//   (this object) <-> TcCOM Objects/XTS ProcessingUnit 1/XL Part 2/XL Module 50
//     Box 62 (AT5100-0100)/DRV Commutation angle/Commutation angle <-> Data Pointer/CommutationAngle
//     Box 62 (AT5100-0100)/DRV Controlword/Controlword <-> Data Pointer/Control
//     Box 62 (AT5100-0100)/DRV Statusword/Statusword <-> Data Pointer/Status
//     Box 62 (AT5100-0100)/DRV Target torque/Target torque <-> Data Pointer/Torque
//     Box 62 (AT5100-0100)/DRV Torque actual value/Torque actual value <-> Data Pointer/ActTorque
//     Box 62 (AT5100-0100)/XFB Inputs/Data <-> Data Pointer/HallSensorValues
//   (this object) <-> TcCOM Objects/XTS ProcessingUnit 1/XL Part 2/XL Module 51
//     Box 63 (AT5100-0100)/DRV Commutation angle/Commutation angle <-> Data Pointer/CommutationAngle
//     Box 63 (AT5100-0100)/DRV Controlword/Controlword <-> Data Pointer/Control
//     Box 63 (AT5100-0100)/DRV Statusword/Statusword <-> Data Pointer/Status
//     Box 63 (AT5100-0100)/DRV Target torque/Target torque <-> Data Pointer/Torque
//     Box 63 (AT5100-0100)/DRV Torque actual value/Torque actual value <-> Data Pointer/ActTorque
//     Box 63 (AT5100-0100)/XFB Inputs/Data <-> Data Pointer/HallSensorValues
//   (this object) <-> TcCOM Objects/XTS ProcessingUnit 1/XL Part 2/XL Module 52
//     Box 64 (AT5100-0100)/DRV Commutation angle/Commutation angle <-> Data Pointer/CommutationAngle
//     Box 64 (AT5100-0100)/DRV Controlword/Controlword <-> Data Pointer/Control
//     Box 64 (AT5100-0100)/DRV Statusword/Statusword <-> Data Pointer/Status
//     Box 64 (AT5100-0100)/DRV Target torque/Target torque <-> Data Pointer/Torque
//     Box 64 (AT5100-0100)/DRV Torque actual value/Torque actual value <-> Data Pointer/ActTorque
//     Box 64 (AT5100-0100)/XFB Inputs/Data <-> Data Pointer/HallSensorValues
//   (this object) <-> TcCOM Objects/XTS ProcessingUnit 1/XL Part 2/XL Module 53
//     Box 65 (AT5100-0100)/DRV Commutation angle/Commutation angle <-> Data Pointer/CommutationAngle
//     Box 65 (AT5100-0100)/DRV Controlword/Controlword <-> Data Pointer/Control
//     Box 65 (AT5100-0100)/DRV Statusword/Statusword <-> Data Pointer/Status
//     Box 65 (AT5100-0100)/DRV Target torque/Target torque <-> Data Pointer/Torque
//     Box 65 (AT5100-0100)/DRV Torque actual value/Torque actual value <-> Data Pointer/ActTorque
//     Box 65 (AT5100-0100)/XFB Inputs/Data <-> Data Pointer/HallSensorValues
//   (this object) <-> TcCOM Objects/XTS ProcessingUnit 1/XL Part 2/XL Module 54
//     Box 66 (AT5100-0100)/DRV Commutation angle/Commutation angle <-> Data Pointer/CommutationAngle
//     Box 66 (AT5100-0100)/DRV Controlword/Controlword <-> Data Pointer/Control
//     Box 66 (AT5100-0100)/DRV Statusword/Statusword <-> Data Pointer/Status
//     Box 66 (AT5100-0100)/DRV Target torque/Target torque <-> Data Pointer/Torque
//     Box 66 (AT5100-0100)/DRV Torque actual value/Torque actual value <-> Data Pointer/ActTorque
//     Box 66 (AT5100-0100)/XFB Inputs/Data <-> Data Pointer/HallSensorValues
//   (this object) <-> TcCOM Objects/XTS ProcessingUnit 1/XL Part 2/XL Module 55
//     Box 67 (AT5100-0100)/DRV Commutation angle/Commutation angle <-> Data Pointer/CommutationAngle
//     Box 67 (AT5100-0100)/DRV Controlword/Controlword <-> Data Pointer/Control
//     Box 67 (AT5100-0100)/DRV Statusword/Statusword <-> Data Pointer/Status
//     Box 67 (AT5100-0100)/DRV Target torque/Target torque <-> Data Pointer/Torque
//     Box 67 (AT5100-0100)/DRV Torque actual value/Torque actual value <-> Data Pointer/ActTorque
//     Box 67 (AT5100-0100)/XFB Inputs/Data <-> Data Pointer/HallSensorValues
//   (this object) <-> TcCOM Objects/XTS ProcessingUnit 1/XL Part 2/XL Module 56
//     Box 68 (AT5100-0100)/DRV Commutation angle/Commutation angle <-> Data Pointer/CommutationAngle
//     Box 68 (AT5100-0100)/DRV Controlword/Controlword <-> Data Pointer/Control
//     Box 68 (AT5100-0100)/DRV Statusword/Statusword <-> Data Pointer/Status
//     Box 68 (AT5100-0100)/DRV Target torque/Target torque <-> Data Pointer/Torque
//     Box 68 (AT5100-0100)/DRV Torque actual value/Torque actual value <-> Data Pointer/ActTorque
//     Box 68 (AT5100-0100)/XFB Inputs/Data <-> Data Pointer/HallSensorValues
//   (this object) <-> TcCOM Objects/XTS ProcessingUnit 1/XL Part 2/XL Module 57
//     Box 69 (AT5100-0100)/DRV Commutation angle/Commutation angle <-> Data Pointer/CommutationAngle
//     Box 69 (AT5100-0100)/DRV Controlword/Controlword <-> Data Pointer/Control
//     Box 69 (AT5100-0100)/DRV Statusword/Statusword <-> Data Pointer/Status
//     Box 69 (AT5100-0100)/DRV Target torque/Target torque <-> Data Pointer/Torque
//     Box 69 (AT5100-0100)/DRV Torque actual value/Torque actual value <-> Data Pointer/ActTorque
//     Box 69 (AT5100-0100)/XFB Inputs/Data <-> Data Pointer/HallSensorValues
//   (this object) <-> TcCOM Objects/XTS ProcessingUnit 1/XL Part 3/XL Module 1
//     Box 74 (AT5100-0100)/DRV Commutation angle/Commutation angle <-> Data Pointer/CommutationAngle
//     Box 74 (AT5100-0100)/DRV Controlword/Controlword <-> Data Pointer/Control
//     Box 74 (AT5100-0100)/DRV Statusword/Statusword <-> Data Pointer/Status
//     Box 74 (AT5100-0100)/DRV Target torque/Target torque <-> Data Pointer/Torque
//     Box 74 (AT5100-0100)/DRV Torque actual value/Torque actual value <-> Data Pointer/ActTorque
//     Box 74 (AT5100-0100)/XFB Inputs/Data <-> Data Pointer/HallSensorValues
//   (this object) <-> TcCOM Objects/XTS ProcessingUnit 1/XL Part 3/XL Module 2
//     Box 75 (AT5100-0100)/DRV Commutation angle/Commutation angle <-> Data Pointer/CommutationAngle
//     Box 75 (AT5100-0100)/DRV Controlword/Controlword <-> Data Pointer/Control
//     Box 75 (AT5100-0100)/DRV Statusword/Statusword <-> Data Pointer/Status
//     Box 75 (AT5100-0100)/DRV Target torque/Target torque <-> Data Pointer/Torque
//     Box 75 (AT5100-0100)/DRV Torque actual value/Torque actual value <-> Data Pointer/ActTorque
//     Box 75 (AT5100-0100)/XFB Inputs/Data <-> Data Pointer/HallSensorValues
//   (this object) <-> TcCOM Objects/XTS ProcessingUnit 1/XL Part 3/XL Module 3
//     Box 76 (AT5100-0100)/DRV Commutation angle/Commutation angle <-> Data Pointer/CommutationAngle
//     Box 76 (AT5100-0100)/DRV Controlword/Controlword <-> Data Pointer/Control
//     Box 76 (AT5100-0100)/DRV Statusword/Statusword <-> Data Pointer/Status
//     Box 76 (AT5100-0100)/DRV Target torque/Target torque <-> Data Pointer/Torque
//     Box 76 (AT5100-0100)/DRV Torque actual value/Torque actual value <-> Data Pointer/ActTorque
//     Box 76 (AT5100-0100)/XFB Inputs/Data <-> Data Pointer/HallSensorValues
//   (this object) <-> TcCOM Objects/XTS ProcessingUnit 1/XL Part 3/XL Module 4
//     Box 77 (AT5100-0100)/DRV Commutation angle/Commutation angle <-> Data Pointer/CommutationAngle
//     Box 77 (AT5100-0100)/DRV Controlword/Controlword <-> Data Pointer/Control
//     Box 77 (AT5100-0100)/DRV Statusword/Statusword <-> Data Pointer/Status
//     Box 77 (AT5100-0100)/DRV Target torque/Target torque <-> Data Pointer/Torque
//     Box 77 (AT5100-0100)/DRV Torque actual value/Torque actual value <-> Data Pointer/ActTorque
//     Box 77 (AT5100-0100)/XFB Inputs/Data <-> Data Pointer/HallSensorValues
//   (this object) <-> TcCOM Objects/XTS ProcessingUnit 1/XL Part 3/XL Module 46
//     Box 72 (AT5100-0100)/DRV Commutation angle/Commutation angle <-> Data Pointer/CommutationAngle
//     Box 72 (AT5100-0100)/DRV Controlword/Controlword <-> Data Pointer/Control
//     Box 72 (AT5100-0100)/DRV Statusword/Statusword <-> Data Pointer/Status
//     Box 72 (AT5100-0100)/DRV Target torque/Target torque <-> Data Pointer/Torque
//     Box 72 (AT5100-0100)/DRV Torque actual value/Torque actual value <-> Data Pointer/ActTorque
//     Box 72 (AT5100-0100)/XFB Inputs/Data <-> Data Pointer/HallSensorValues
//   (this object) <-> TcCOM Objects/XTS ProcessingUnit 1/XL Part 3/XL Module 47
//     Box 73 (AT5100-0100)/DRV Commutation angle/Commutation angle <-> Data Pointer/CommutationAngle
//     Box 73 (AT5100-0100)/DRV Controlword/Controlword <-> Data Pointer/Control
//     Box 73 (AT5100-0100)/DRV Statusword/Statusword <-> Data Pointer/Status
//     Box 73 (AT5100-0100)/DRV Target torque/Target torque <-> Data Pointer/Torque
//     Box 73 (AT5100-0100)/DRV Torque actual value/Torque actual value <-> Data Pointer/ActTorque
//     Box 73 (AT5100-0100)/XFB Inputs/Data <-> Data Pointer/HallSensorValues
//   (this object) <-> TcCOM Objects/XTS ProcessingUnit 1/XL Part 3/XL Module 5
//     Box 78 (AT5100-0100)/DRV Commutation angle/Commutation angle <-> Data Pointer/CommutationAngle
//     Box 78 (AT5100-0100)/DRV Controlword/Controlword <-> Data Pointer/Control
//     Box 78 (AT5100-0100)/DRV Statusword/Statusword <-> Data Pointer/Status
//     Box 78 (AT5100-0100)/DRV Target torque/Target torque <-> Data Pointer/Torque
//     Box 78 (AT5100-0100)/DRV Torque actual value/Torque actual value <-> Data Pointer/ActTorque
//     Box 78 (AT5100-0100)/XFB Inputs/Data <-> Data Pointer/HallSensorValues
//   (this object) <-> TcCOM Objects/XTS ProcessingUnit 1/XL Part 3/XL Module 6
//     Box 79 (AT5100-0100)/DRV Commutation angle/Commutation angle <-> Data Pointer/CommutationAngle
//     Box 79 (AT5100-0100)/DRV Controlword/Controlword <-> Data Pointer/Control
//     Box 79 (AT5100-0100)/DRV Statusword/Statusword <-> Data Pointer/Status
//     Box 79 (AT5100-0100)/DRV Target torque/Target torque <-> Data Pointer/Torque
//     Box 79 (AT5100-0100)/DRV Torque actual value/Torque actual value <-> Data Pointer/ActTorque
//     Box 79 (AT5100-0100)/XFB Inputs/Data <-> Data Pointer/HallSensorValues
//   (this object) <-> TcCOM Objects/XTS ProcessingUnit 1/XL Part 3/XL Module 7
//     Box 80 (AT5100-0100)/DRV Commutation angle/Commutation angle <-> Data Pointer/CommutationAngle
//     Box 80 (AT5100-0100)/DRV Controlword/Controlword <-> Data Pointer/Control
//     Box 80 (AT5100-0100)/DRV Statusword/Statusword <-> Data Pointer/Status
//     Box 80 (AT5100-0100)/DRV Target torque/Target torque <-> Data Pointer/Torque
//     Box 80 (AT5100-0100)/DRV Torque actual value/Torque actual value <-> Data Pointer/ActTorque
//     Box 80 (AT5100-0100)/XFB Inputs/Data <-> Data Pointer/HallSensorValues
//   (this object) <-> TcCOM Objects/XTS ProcessingUnit 1/XL Part 3/XL Module 8
//     Box 81 (AT5100-0100)/DRV Commutation angle/Commutation angle <-> Data Pointer/CommutationAngle
//     Box 81 (AT5100-0100)/DRV Controlword/Controlword <-> Data Pointer/Control
//     Box 81 (AT5100-0100)/DRV Statusword/Statusword <-> Data Pointer/Status
//     Box 81 (AT5100-0100)/DRV Target torque/Target torque <-> Data Pointer/Torque
//     Box 81 (AT5100-0100)/DRV Torque actual value/Torque actual value <-> Data Pointer/ActTorque
//     Box 81 (AT5100-0100)/XFB Inputs/Data <-> Data Pointer/HallSensorValues

CONFIGURATION PlanarTrackMovement_1
    RESOURCE PLC ON TwinCAT3
        TASK PlcTask(INTERVAL := T#2ms, PRIORITY := 20);
        PROGRAM MAIN WITH PlcTask : MAIN;
    END_RESOURCE
END_CONFIGURATION

// ---- DUTs/E_EcState.TcDUT
{attribute 'qualified_only'}
{attribute 'strict'}
{attribute 'to_string'}
TYPE E_EcState :
(
	InitNoCom_Fault := 0,
	Init := 1,
	Preop := 2,
	Boot := 3,
	SafeOP := 4,
	Op_Ready := 8
)UINT := InitNoCom_Fault ;
END_TYPE

// ---- DUTs/E_MergeMode.TcDUT
{attribute 'qualified_only'}
{attribute 'strict'}
TYPE E_MergeMode :
(
	BlockedWait := 0,
	Follow := 1,
	Lead := 2
);
END_TYPE

// ---- DUTs/E_SwitchOpMode.TcDUT
{attribute 'qualified_only'}
//{attribute 'strict'}
TYPE E_SwitchOpMode :
(
  DivertSpecifiedCount	:= 0,
  DivertAll	:= 1
);
END_TYPE

// ---- DUTs/E_TrackNum.TcDUT
{attribute 'qualified_only'}
{attribute 'strict'}
TYPE e_TrackNum :
	(
	Main   :=1,
	Small  :=2,
	Big    :=3
	);	
END_TYPE

// ---- DUTs/MoverSort.TcDUT
TYPE MoverSort :
STRUCT
	MoverNumber 	: UDINT;
	TrackID  		: PlanarTrackOTCID;
	MoverPos 		: LREAL;
	MoverTrackNr 	: UDINT;
END_STRUCT
END_TYPE

// ---- DUTs/ST_Color_Code.TcDUT
TYPE ST_Color_Code :
STRUCT
	Pattern : UINT;
	Red :USINT;
	Green: USINT;
	Blue : USINT; 
END_STRUCT
END_TYPE

// ---- DUTs/ST_DivertConfig.TcDUT
TYPE ST_DivertConfig :
STRUCT
 	SwitchOpMode         						: E_SwitchOpMode;
	IntervalToDivert							: UDINT := 1;
	MaxAllowedDivertCount						: UDINT := 0;
	CurrentFunctionCoeffA						: LREAL := 0.5;
	CurrentFunctionCoeffB						: LREAL := 0.3;
	CurrentFunctionCoeffC						: LREAL := 5.5;
END_STRUCT
END_TYPE;

// ---- DUTs/ST_MergeConfig.TcDUT
TYPE ST_MergeConfig :
STRUCT
	gapStart: LREAL := 5600;
	gapLength: LREAL := 2000;
	moverInFront: UDINT;
	mover1FollowDist: LREAL;
	followSyncPos: LREAL;
	masterSyncPos: LREAL;
	masterPosAtSync: LREAL;
	followerPosAtSync: LREAL;
END_STRUCT
END_TYPE;

// ---- DUTs/ST_MoverConfig.TcDUT
TYPE ST_MoverConfig EXTENDS ST_MoveOnTrackOptions:
STRUCT
	Velo			: LREAL := 1500;
	Accel			: LREAL := 4000;
	Decel			: LREAL := 4000;
	Jerk			: LREAL := 16000;
	VeloComp		: LREAL := 200;
	MoverGap		: LREAL := 900;
END_STRUCT
END_TYPE

// ---- DUTs/ST_PlanarTrackConfig.TcDUT
TYPE ST_PlanarTrackConfig :
STRUCT
	TrackIndex					: E_TrackNum;
	MCTrack						: CDT_MCTOPLC_PLANAR_TRACK;
END_STRUCT
END_TYPE

// ---- DUTs/ST_StaticSectorStatus.TcDUT
TYPE ST_StaticSectorStatus :
STRUCT
	MoverIsOnSector			: BOOL;
	MoverCountOnSector		: UDINT;
	MoverEnteredSector		: Tc2_Standard.R_TRIG;
	MoverExitedSector		: Tc2_Standard.F_TRIG;
	SectorLength				: LREAL;
	MoverDistanceFromEnd	: LREAL;
END_STRUCT
END_TYPE

// ---- DUTs/ST_SwitchConfig.TcDUT
TYPE ST_SwitchConfig :
STRUCT
	MagnetStartPosition				    	    : LREAL := 9850; // mm
	MagnetEndPosition				    	    : LREAL := 10600; // mm
	OnInnerLoopOffMagnetPosn					: LREAL	:= 170; //mm
	SwitchCurrentNominal						: LREAL := 5.8; // A (See function for computation)
	CurrentMultFactor							: LREAL := 1310; // Scaling factor for 10V output=25.0A
    UseNominalCurrentVeloSetpoints              : BOOL;
    UseNominalPositionCoeff			            : BOOL := TRUE;
 	DivertConfig	       						: ST_DivertConfig;
END_STRUCT
END_TYPE;

// ---- DUTs/ST_SwitchStatus.TcDUT
TYPE ST_SwitchStatus :
STRUCT
 	MagnetValue		        AT%Q* 	: INT;
	MagnetEnabled     	        	: BOOL;
    CurrentOutputActual             : LREAL;
    CurrentTheorOutputMax           : LREAL;
	CurrentActualOutput				: LREAL;
    PosnCurrentCoeff                : LREAL;
	ShuttleCountAtDivertTrig		: UDINT;
	ShuttleQueueCount				: UDINT;
	ShuttleCountOnShortcut			: UDINT;
END_STRUCT
END_TYPE

// ---- XlMover/DUTs/DUT.TcDUT
TYPE ST_XtsCommandFeedback :
STRUCT
		(* Returns wether the execution of the method is done. *)
		IsDone : BOOL;
		(* Returns wether the execution of the method is busy. *)
		IsBusy : BOOL;
		(* Returns wether the execution of the method is busy. *)
		HasError : BOOL;
		(* Returns the HRESULT to the call. *)
		{attribute 'GUID' := '18071995-0000-0000-0000-000000000019'}
		{attribute 'GlobalType'}
		HRESULT : GLOBAL.HRESULT;
	END_STRUCT
END_TYPE

// ---- GVLs/GVL_Mc.TcGVL

VAR_GLOBAL PERSISTENT
	nNumMovers			: UINT := 16;
END_VAR


VAR_GLOBAL CONSTANT
	nMoverCount					: UINT := 16;
	nTrackCount					: UINT := 3;
	gciNumStations 				: UINT := 3;
	XtsShortcutOid				: otcid := 16#01010480 ;
	XtsOutterLoopOid 			: otcid := 16#01010490;
END_VAR

VAR_GLOBAL
	//Track_BigCircle		: 	MC_PlanarTrack; 	
	//Track_MainCircle	: 	MC_PlanarTrack;
 	//Track_SmallCircle	: 	MC_PlanarTrack;
	
	MC_Tracks    		:	ARRAY[1..nTrackCount] OF MC_PlanarTrack;
	MC_Trackfeedback	:	ARRAY[1..nTrackCount] OF MC_PlanarFeedback;
	TrackTrail 			:	MC_PlanarTrackTrail;
	
	fbXtsEnvironment			: 	FB_XtsEnvironment;
	ipXlMover 					: 	I_XtsXlMover1;
	ipXtsProcessingUnit			:   I_XtsProcessingUnit1;
	cmdFeedback					: 	XtsCommandFeedback;
	fbMover				:	ARRAY[1..nMoverCount] OF FB_Mover;
	iMover				:	ARRAY[1..nMoverCount] OF I_Mover;
	//fbPlanarMover		:	ARRAY[1..nNumMaxMovers] OF FB_PlanarMover;
	MoverFeedback		:	ARRAY[1..nMoverCount] OF MC_PlanarFeedback;
	aStopPositions : ARRAY [1..nMoverCount] OF LREAL;// := [2400, 1700, 1000, 300];
	
	
	Mover				:	ARRAY[0..nMoverCount] OF MoverSort;
	
	HWStart		AT%I* : BOOL;
	HWStop		AT%I* : BOOL;	
	StartLight 	AT%Q* : BOOL;
	StopLight	AT%Q* : BOOL;
	
	sGraphCalciFrame : T_MaxString := 'https://www.desmos.com/calculator';
END_VAR

// ---- XlMover/ITFs/I_Mover.TcIO

INTERFACE I_Mover

METHOD CycleUpdate : BOOL
VAR_INPUT
END_VAR
END_METHOD

PROPERTY distToEndOfTrack : Lreal
GET
END_GET
END_PROPERTY

METHOD Init : BOOL
VAR_INPUT
	XtsMover:  I_XtsXlMover1;
	XtsProcessingUnit :  I_XtsProcessingUnit1;
END_VAR
END_METHOD

METHOD JoinNearestTrack : BOOL


VAR

END_VAR
END_METHOD

METHOD LeaveSystemAt : BOOL
VAR_INPUT
	ConnectionOut: REFERENCE TO MC_PlanarTrackConnectionOut;	
END_VAR
END_METHOD

METHOD MoveOnTrack : BOOL
VAR_INPUT
	track: REFERENCE TO MC_PlanarTrack;	
	targetPos: LREAL;
	gap : LREAL; 
	velo : LREAL; 
END_VAR
END_METHOD

PROPERTY MoverOTCID : OTCID
GET
END_GET
SET
END_SET
END_PROPERTY

PROPERTY MoverStopped : BOOL
GET
END_GET
SET
END_SET
END_PROPERTY

PROPERTY P_Dynamics : REFERENCE TO DynamicConstraint_PathXY;
GET
END_GET
END_PROPERTY

PROPERTY P_IsInitialized : bool
GET
END_GET
END_PROPERTY

PROPERTY P_PlanarFeedback : REFERENCE TO MC_PlanarFeedback
GET
END_GET
END_PROPERTY

PROPERTY P_PlanarMover :   REFERENCE TO  MC_PlanarMover
GET
END_GET
END_PROPERTY

PROPERTY P_SyncFeedback :  REFERENCE TO MC_PlanarFeedbackGearInPosOnTrackWithMasterMover
GET
END_GET
END_PROPERTY

PROPERTY P_TargetTrack : UDINT
GET
END_GET
SET
END_SET
END_PROPERTY

PROPERTY Rework : BOOL
GET
END_GET
SET
END_SET
END_PROPERTY

METHOD SyncToOtherMover : Bool
VAR_INPUT
	masterSyncPos : LREAL; // Position on the master track
	followerSyncPos : LREAL; // position on the follower track
	PlanarMoverToFollow: REFERENCE TO Tc3_Mc3PlanarMotion.MC_PlanarMover;
	masterTrack : REFERENCE TO Tc3_Mc3PlanarMotion.MC_PlanarTrack; 
	followerTrack : REFERENCE TO Tc3_Mc3PlanarMotion.MC_PlanarTrack; 
	velo :  REFERENCE TO LREAL; 
END_VAR
END_METHOD

METHOD  UpdateXtsTrack
VAR_INPUT
END_VAR
VAR

END_VAR
END_METHOD

PROPERTY XlProcessingUnit : I_XtsProcessingUnit1
GET
END_GET
END_PROPERTY

PROPERTY XtsComFeed : REFERENCE TO  XtsCommandFeedback
GET
END_GET
END_PROPERTY

PROPERTY XtsXlMover :  I_XtsXlMover1
GET
END_GET
END_PROPERTY

END_INTERFACE

// ---- POUs/MAIN.TcPOU
PROGRAM MAIN
VAR

	bAllDone		: BOOL;
	bStopSequence	: BOOL;
	HMI_StopCmd		: BOOL;
	
	nCase 		: INT;
	nMoveState		: ARRAY[1..nMoverCount] OF INT;
	

	
	nForCounter: UDINT;
	M,N,T,Tr : UINT;
//	slowDynamics: DynamicConstraint_PathXY;
	haltDynamics : DynamicConstraint_PathXY;
	stopAndWait : ARRAY[1..GVL_Mc.nMoverCount] OF TON; 
	waitForGapParkPos: LREAL := 3500;
	// Magnet
	MagnetValue AT%Q*: INT;
	MagnetFdbkValue AT%I* : INT;
	bMagnetOn : BOOL;	

	Init : BOOL ; 	
	
	IsMoverCommandedInShortcut: BOOL;
	IsMoverInBlockingArea: BOOL;
	nActStopPos: UINT := 1;
	Fp_error : R_Trig;

	Switch : BOOL;
	WithoutSwitch : BOOL := TRUE;
	SwtichOnly: BOOL;
	
	MoverStop 	AT%I* :BOOL;
	MoverStopDone AT%Q*		: BOOL;
	Info 		AT%Q*: BOOL;
	Operating	AT%Q*: BOOL;
	Process		AT%Q*: BOOL;
	Fault		AT%Q*: BOOL;
	Emergency	AT%Q*: BOOL;
	
	Voltage1 AT%I*: UDINT;
	Voltage2 AT%I*: UDINT;
	
	
	TcRestart : TC_Restart;
	Restart : BOOL;
	busy : BOOL;
	rt_InitStart : R_TRIG;
	rt_InitStop : R_TRIG;
	bStartSequence: BOOL;
	
	FP_Counter : r_trig;
	Switchcounter : DINT;
	test : LREAL;
	Horntimer : tp; 
	R_trigHorn : R_trig;
	
	TestPowerMat : BOOL := TRUE;
	StopTime : TIME := T#1S;
	StopTimer :ARRAY[1..nMoverCount] OF ton;
	StartTimer :ARRAY[1..nMoverCount] OF BOOL;
	
	
	MoverPos :ARRAY[1..nMoverCount] OF PositionXYC;
	ArcLength :ARRAY[1..nMoverCount] OF LREAL;
	TrackPos :ARRAY[1..nMoverCount] OF ARRAY[1..nMoverCount] OF PositionXYC;
	
	//searchGap : F_SearchTheBigTrackForAHole; 
	aMoverTrack : ARRAY[1..nMoverCount] OF Global.OTCID;
	FirstMoverTrackPos : LREAL;
	MoverGap : LREAL;
	FTrigTrackCount : F_Trig;
	MoverNo  : UDINT;
	stMoverConfigSlow	: ST_MoverConfig;
	stMoverConfigNormal : ST_MoverConfig;
	stMoverConfigFast  : ST_MoverConfig;
	stMoverCfgAggressive : ST_MoverConfig;
	stMoverCfgHalt : ST_MoverConfig;
	
	stMergeConfig		 : ST_MergeConfig;
	SwitchConfig		 : ST_SwitchConfig;
	
	SwitchStatus 		  : ST_SwitchStatus;

	ModuleState1 AT%I*: E_EcState;
	ModuleState2 AT%I*: E_EcState;
	ModuleState3 AT%I*: ARRAY[0..2] OF E_EcState;
	
	MessageTrigger : ARRAY[1..20] OF R_trig;
	
	//========= Merge =========================================
	
	SwitchParkPos : LREAL := 3500;
	nextMoverForSwitch: UDINT :=1;
	moverInSwitchDoNotSendAnother: BOOL;
	trapError: BOOL;
	trapErrorID: UDINT;
	moverWithFault: UDINT;
	stepWithFault: INT;
	
	followSyncPos: LREAL;
	masterSyncPos: LREAL;
	masterPosAtSync: LREAL;
	followerPosAtSync: LREAL;
	moverInFront: UDINT;
	gapStart: LREAL := 8500; //5600
	gapLength: LREAL := 2200; //1800
	fbTrackobject : FB_TrackObject;
	getList: BOOL;
	directMerge: BOOL;
	mergeNotPossible: BOOL;
	
	endOfBigTrack : LREAL; 
	endOfSmallTrack : LREAL; 
	endOfMainTrack : LREAL; 
	followerToEndOfTrack: LREAL;
	leaderToEndofTrack: LREAL;
	distToMoverInFront: LREAL;
END_VAR


// =====================
// Initalize XTS Utility
GVL_MC.fbXtsEnvironment.Init(GVL_MC.cmdFeedback);
IF NOT GVL_MC.cmdFeedback.IsDone THEN
	RETURN;
END_IF
//*****************************************************
Emergency :=  MoverStop;

Operating := NOT  MoverStop;

//================== Check Voltage=====================================================
R_trigHorn(clk := Voltage1< 250000 );
//Horntimer(in:= ( R_trigHorn.Q ) , PT:= T#2S,Q=> info);
IF R_trigHorn.Q THEN
	ADSLOGSTR(msgCtrlMask:= ADSLOG_MSGTYPE_LOG , msgFmtStr:= 'Module Voltage Fault ' , strArg:= '');
END_IF 
//=================== Check State of Modules===========================================

MessageTrigger[1](clk:=ModuleState1 <> 8 AND nCASE> 0);
IF MessageTrigger[1].Q THEN
	ADSLOGSTR(msgCtrlMask:= ADSLOG_MSGTYPE_LOG , msgFmtStr:= 'Module Fault Line 1 %s' , strArg:= TO_STRING(ModuleState1));
END_IF

MessageTrigger[2](clk:=ModuleState2 <> 8 AND nCASE> 0);
IF MessageTrigger[2].Q THEN
	ADSLOGSTR(msgCtrlMask:= ADSLOG_MSGTYPE_LOG , msgFmtStr:= 'Module Fault Line 2 %s ' , strArg:= TO_STRING(ModuleState2));
END_IF

MessageTrigger[3](clk:=ModuleState3[0] <> 8 AND nCASE> 0);
IF MessageTrigger[3].Q THEN
	ADSLOGSTR(msgCtrlMask:= ADSLOG_MSGTYPE_LOG , msgFmtStr:= 'Module Fault Line 3 Default SyncUnit %s ' , strArg:= TO_STRING(ModuleState3[0]));
END_IF

MessageTrigger[4](clk:=ModuleState3[1] <> 8 AND nCASE> 0);
IF MessageTrigger[4].Q THEN
	ADSLOGSTR(msgCtrlMask:= ADSLOG_MSGTYPE_LOG , msgFmtStr:= 'Module Fault Line 3 XtsTask SyncUnit %s ' , strArg:= TO_STRING(ModuleState3[1]));
END_IF

MessageTrigger[5](clk:=ModuleState3[2] <> 8 AND nCASE> 0);
IF MessageTrigger[5].Q THEN
	ADSLOGSTR(msgCtrlMask:= ADSLOG_MSGTYPE_LOG , msgFmtStr:= 'Module Fault Line 3 PlcTask SyncUnit %s ' , strArg:= TO_STRING(ModuleState3[2]));
END_IF

//=====================================================================================

IF nCASE > 90 THEN
	Process := TRUE;
ELSE 
	Process := FALSE;	
END_IF

IF NOT MoverStop AND NOT MoverStopDone THEN
	ADSLOGSTR(msgCtrlMask:= ADSLOG_MSGTYPE_LOG , msgFmtStr:= 'E-Stop ' , strArg:= '');
	FOR nForCounter:=1 TO nNumMovers DO
		fbMover[nForCounter].P_Dynamics.SetValuesVADJ(stMoverConfigNormal.velo,stMoverConfigNormal.Accel,stMoverConfigNormal.Decel,stMoverConfigNormal.Jerk);
		nCase := 140;
	END_FOR		
	MoverStopDone := TRUE;
ELSIF 	MoverStop THEN
	MoverStopDone := FALSE;
END_IF



TcRestart(
NETID:= '', 
RESTART:= Restart OR (GVL_Mc.HWStart AND NOT GVL_Mc.HWStop), 
TMOUT:=T#5S , 
BUSY=>busy , 
ERR=> , 
ERRID=> );

rt_InitStart(clk:= (bStartSequence OR GVL_Mc.HWStart) AND GVL_Mc.HWStop);
IF rt_InitStart.Q THEN
	nCase := 10;
	bStartSequence	:= FALSE;

	stMoverConfigSlow.Velo := 1000;
// 	stMoverConfigSlow.Accel := 4000;
// 	stMoverConfigSlow.Decel := 4000; 
// 	stMoverConfigSlow.Jerk := 16000;
	stMoverConfigFast.Velo := 4000;
// 	stMoverConfigFast.Accel := 4000;
// 	stMoverConfigFast.Decel := 4000; 
// 	stMoverConfigFast.Jerk := 16000;
	stMoverCfgHalt.Decel := 3000; 
	stMoverCfgHalt.Jerk := 24000;
	
//	slowDynamics.SetValuesVADJ(stMoverConfigSlow.Velo,stMoverConfigSlow.Accel,stMoverConfigSlow.Decel,stMoverConfigSlow.Jerk);
//	fastDynamics.SetValuesVADJ(stMoverConfigFast.Velo,stMoverConfigFast.Accel,stMoverConfigFast.Decel,stMoverConfigFast.Jerk);
	haltDynamics.SetValuesVADJ(stMoverCfgHalt.Velo,stMoverCfgHalt.Accel,stMoverCfgHalt.Decel,stMoverCfgHalt.Jerk);
END_IF
	haltDynamics.SetValuesVADJ(stMoverCfgHalt.Velo,stMoverCfgHalt.Accel,stMoverCfgHalt.Decel,stMoverCfgHalt.Jerk);
GVL_Mc.StartLight := MoverStop AND nCase < 100;
GVL_Mc.StopLight  := (nCase = 100);

IsMoverInBlockingArea := FALSE;

FOR M := 1 TO GVL_Mc.nNumMovers DO///Movers
	StopTimer[M](in:=StartTimer[m],PT:=StopTime);

	
	IF NOT GVL_MC.fbMover[GVL_Mc.nNumMovers].P_IsInitialized THEN
		GVL_MC.ipXtsProcessingUnit :=  GVL_MC.fbXtsEnvironment.ProcessingUnit(1,0);
		GVL_MC.ipXlMover  :=  GVL_MC.fbXtsEnvironment.ProcessingUnit(1, 0).XlMover(m, 0);
		GVL_MC.fbMover[m].Init( GVL_MC.ipXlMover, GVL_MC.ipXtsProcessingUnit); 
		iMover[m] := fbMover[m] ;
	END_IF
	 MoverFeedback[m].Update();
	GVL_MC.fbMover[m].CycleUpdate();
	
	GVL_Mc.Mover[M].MoverPos  :=GVL_MC.fbMover[M].P_PlanarMover.MCTOPLC.SETONTRACK.SetPos;
	GVL_Mc.Mover[M].TrackID:= GVL_MC.fbMover[M].P_PlanarMover.MCTOPLC.SETONTRACK.TrackOID;
	GVL_Mc.Mover[M].MoverNumber := M;
		
	TR := Tr+1;
	IF Tr = 4 THEN
		Tr :=1;
	END_IF
	ArcLength[M] :=GVL_Mc.MC_Tracks[Tr].GetArcLengthClosestTo(MoverPos[M]);
	GVL_Mc.MC_Tracks[Tr].GetPositionAt(ArcLength[M],TrackPos[M][Tr]);
	
	IF ABS(MoverPos[m].x - TrackPos[M][Tr].x) < 1 AND  ABS(MoverPos[m].y - TrackPos[M][Tr].y) < 1 THEN
 		GVL_Mc.Mover[M].MoverTrackNr := Tr;
	END_IF	
	
	IsMoverInBlockingArea := IsMoverInBlockingArea OR (Mover[M].TrackID = GVL_Mc.MC_Tracks[E_TrackNum.main].MCTOPLC_STD.TrackOID AND IsBetween(Mover[M].MoverPos, SwitchConfig.MagnetStartPosition - 100, SwitchConfig.MagnetEndPosition + 100));

	Fp_error(clk := GVL_MC.fbMover[M].P_PlanarMover.Error AND GVL_MC.fbMover[M].XtsXlMover.GetIsActive(0) AND nCASE = 100);
	IF Fp_error.Q THEN
		nCase := 140;
		Fault := TRUE;
		bMagnetOn := FALSE;
		ADSLOGSTR(msgCtrlMask:= ADSLOG_MSGTYPE_LOG , msgFmtStr:= 'Mover %s Faulted ' , strArg:= INT_TO_STRING(M));
	ELSE
		Fault := FALSE;
	END_IF
	
	IF aMoverTrack[1] <> 0 AND_THEN GVL_MC.fbMover[M].P_PlanarMover.MCTOPLC.STD.MoverOID = aMoverTrack[1] THEN
		FirstMoverTrackPos := GVL_MC.fbMover[M].P_PlanarMover.MCTOPLC.SETONTRACK.SetPos;
	END_IF
	
END_FOR

FOR T := 1 TO nTrackCount DO 
	MC_Tracks[T].Update();
	MC_Trackfeedback[T].Update();
	
END_FOR
 MoverGap := (GVL_Mc.MC_Tracks[E_TrackNum.Big].GetLength()- FirstMoverTrackPos);
 
//================  merge ===============

fbTrackobject(TrackID:= MC_Tracks[E_TrackNum.big].MCTOPLC_STD.TrackOID,iMover:= iMover,trackLength:= GVL_Mc.MC_Tracks[E_TrackNum.Big].GetLength()); 
fbTrackobject.CyclicUpdate(); 


//======================================

CASE nCase OF
	10:
		
		Fault := FALSE;
		nCase := 20;

	20:
		FOR T := 1 TO nTrackCount DO 
			MC_Tracks[T].Enable(MC_Trackfeedback[T]);
		END_FOR
				nCase := 30;
				
	30: 
		IF MC_Trackfeedback[1].Done AND MC_Trackfeedback[2].Done AND MC_Trackfeedback[3].Done THEN
			nCase := 35;
		END_IF
		
		
	35:
		FOR nForCounter:=1 TO nNumMovers DO
			GVL_MC.fbMover[nForCounter].P_Dynamics.SetValuesVADJ(stMoverConfigNormal.velo,stMoverConfigNormal.Accel,stMoverConfigNormal.Decel,stMoverConfigNormal.Jerk);
			fbMover[nForCounter].P_PlanarMover.Reset(MoverFeedback[nForCounter]);
		END_FOR
		nCase := 36;	
			
	36:	
		bAllDone:=TRUE;
		FOR nForCounter:=1 TO nNumMovers DO
			bAllDone:=bAllDone AND MoverFeedback[nForCounter].Done;
		END_FOR
		
		IF bAllDone THEN
			nCase := 40;
		END_IF
				
	40:
		FOR nForCounter:=1 TO nNumMovers DO
			fbMover[nForCounter].P_PlanarMover.Enable(MoverFeedback[nForCounter]);
		END_FOR
		nCase := 50;
			
	50:
		bAllDone:=TRUE;
		FOR nForCounter:=1 TO nNumMovers DO
			bAllDone:=bAllDone AND MoverFeedback[nForCounter].Done;
		END_FOR
		
		IF bAllDone THEN
			nCase := 60;
		END_IF

	60:
		FOR nForCounter:=nNumMovers TO 1  BY -1 DO
			fbMover[nForCounter].JoinNearestTrack();
		END_FOR
		
		nCase := 70;
		
		
	70:
		bAllDone:=TRUE;
		FOR nForCounter:=1 TO nNumMovers DO
			bAllDone:=bAllDone AND fbMover[nForCounter].P_PlanarFeedback.Done;
		END_FOR
		
		IF bAllDone THEN
			nCase := 80;
		END_IF
		
	80:	
		FOR nForCounter:=1 TO nNumMovers DO
			nMoveState[nForCounter] := 0;
		END_FOR
		
		nCase := 100;

	100:
		
		FOR nForCounter:=1 TO nNumMovers DO
			fbMover[nForCounter].P_Dynamics.SetValuesVADJ(stMoverConfigNormal.velo,stMoverConfigNormal.Accel,stMoverConfigNormal.Decel,stMoverConfigNormal.Jerk);
			IF MoverNo <> 0 AND_THEN 	fbMover[MoverNo].P_PlanarMover.MCTOPLC.SETONTRACK.TrackOID =	 GVL_Mc.MC_Tracks[E_TrackNum.Big].MCTOPLC_STD.TrackOID THEN
				IsMoverCommandedInShortcut := FALSE;
			//	MoverNo := 0;
			END_IF
			
			//Adjust the first mover parameters to induce a platoon
			fbMover[1].P_Dynamics.SetValuesVADJ(V:= stMoverConfigNormal.velo-stMoverConfigNormal.VeloComp, A:= stMoverConfigNormal.Accel, D:= stMoverConfigNormal.Decel, J:= stMoverConfigNormal.Jerk);	
				
			CASE nMoveState[nForCounter] OF
				
				0: // Track 3 Main Cycle
					fbMover[nForCounter].P_Dynamics.SetValuesVADJ(stMoverConfigNormal.velo,stMoverConfigNormal.Accel,stMoverConfigNormal.Decel,stMoverConfigNormal.Jerk);
					fbMover[nForCounter].MoveOnTrack(track:= GVL_Mc.MC_Tracks[E_TrackNum.Main], targetPos:= GVL_Mc.MC_Tracks[E_TrackNum.Main].GetLength()-500, gap:= stMoverConfigNormal.MoverGap, velo:= stMoverConfigNormal.velo);
				
					nMoveState[nForCounter] := 10;
					
				10:
					IF Mover[nForCounter].MoverPos > GVL_Mc.MC_Tracks[E_TrackNum.Main].GetLength()-6000  AND  Mover[nForCounter].TrackID =   GVL_Mc.MC_Tracks[E_TrackNum.Main].MCTOPLC_STD.TrackOID    THEN//     MCTrackOid_MainSemicircle THEN
						IF  (SwtichOnly OR NOT IsMoverCommandedInShortcut )AND NOT WithoutSwitch  AND  nForCounter = nextMoverForSwitch THEN // AND NOT( moverInSwitchDoNotSendAnother)  THEN
							nMoveState[nForCounter] := 40; // 20 - BigCycel
								moverInSwitchDoNotSendAnother := TRUE; 
							//IF fbPlanarMover[nForCounter].IsCommandedInShortcut THEN
								IsMoverCommandedInShortcut := TRUE;
								MoverNo :=nForCounter; /// fbPlanarMover[nForCounter].McPlanarMover.MCTOPLC.STD.MoverOID;
								IF nextMoverForSwitch >= nNumMovers THEN // send the next mover to the switch
									nextMoverForSwitch := 1; 
								ELSE 
									nextMoverForSwitch := nextMoverForSwitch + 1; 
								END_IF
							//END_IF
						ELSE
							nMoveState[nForCounter] := 20;  // 40- SmallCycel					
						END_IF
					END_IF

				
				20:
					fbMover[nForCounter].P_Dynamics.SetValuesVADJ(stMoverConfigNormal.velo,stMoverConfigNormal.Accel,stMoverConfigNormal.Decel,stMoverConfigNormal.Jerk);
					fbMover[nForCounter].MoveOnTrack(track:= GVL_Mc.MC_Tracks[E_TrackNum.Big], targetPos:= GVL_Mc.MC_Tracks[E_TrackNum.Big].GetLength()-1000, gap:= stMoverConfigNormal.MoverGap, velo:= stMoverConfigNormal.velo);
			
					nMoveState[nForCounter] := 30;
				
					
				30:
					IF fbMover[nForCounter].P_PlanarFeedback.Error AND NOT trapError THEN //trap the error once.  
						moverWithFault := nForCounter; 
						trapError := fbMover[nForCounter].P_PlanarFeedback.Error; 
						trapErrorID := fbMover[nForCounter].P_PlanarFeedback.ErrorId; 
						stepWithFault := 30; 
					END_IF 
					IF Mover[nForCounter].MoverPos > GVL_Mc.MC_Tracks[E_TrackNum.Big].GetLength()-10000 AND  Mover[nForCounter].TrackID = GVL_Mc.MC_Tracks[E_TrackNum.big].MCTOPLC_STD.TrackOID    THEN//      MCTrackOid_BigSemicircle THEN
						nMoveState[nForCounter] := 0;
					END_IF				
				
			
				40:
					fbMover[nForCounter].P_Dynamics.SetValuesVADJ(stMoverConfigNormal.velo,stMoverConfigNormal.Accel,stMoverConfigNormal.Decel,stMoverConfigNormal.Jerk);
					fbMover[nForCounter].MoveOnTrack(track:= GVL_Mc.MC_Tracks[E_TrackNum.Small], targetPos:= SwitchParkPos, gap:= stMoverConfigNormal.MoverGap, velo:= stMoverConfigNormal.velo);
					
					nMoveState[nForCounter] := 45;
	
				45: 
					IF fbMover[nForCounter].P_PlanarFeedback.Error AND NOT trapError THEN //trap the error once.   
						trapError := fbMover[nForCounter].P_PlanarFeedback.Error; 
						trapErrorID := fbMover[nForCounter].P_PlanarFeedback.ErrorId;
						stepWithFault := 45;
 						moverWithFault := nForCounter; 
					END_IF
					IF fbMover[nForCounter].P_PlanarFeedback.Done THEN 
						nMoveState[nForCounter] := 50; //50;
						stopAndWait[nForCounter](IN:=TRUE, PT:=StopTime); 
					END_IF 	

				50:
					stopAndWait[nForCounter](); 
					IF stopAndWait[nForCounter].Q  OR NOT TestPowerMat THEN // send the mover to a sync Position 2.6m before the end of the track 
						stopAndWait[nForCounter](IN:=FALSE); 							
					//	fbMover[nForCounter].P_Dynamics.SetValuesVADJ(stMoverConfigNormal.velo,stMoverConfigNormal.Accel,stMoverConfigNormal.Decel,stMoverConfigNormal.Jerk);
					//	fbMover[nForCounter].MoveOnTrack( GVL_Mc.MC_Tracks[E_TrackNum.Small], GVL_Mc.MC_Tracks[E_TrackNum.Small].GetLength()-waitForGapParkPos,stMoverConfigNormal.MoverGap,stMoverConfigNormal.velo);
					//	searchGap(resetSearch:=TRUE, fbMover := fbMover); 
						nMoveState[nForCounter] := 60; 
					END_IF 
					
				60: // look for a merge position 
					//IF fbMover[nForCounter].P_PlanarFeedback.Done THEN// MCTrackOid_Shortcut THEN
							fbTrackobject.findMergePosition(
								mergeSyncCommandPos := gapStart , 
								spaceToMerge := gapLength, 
								nMoverToFollow => moverInFront, 
								mergeWithoutFollow => directMerge, 
								mergeNotPossible => mergeNotPossible); 
							IF directMerge OR  ( moverInFront <> 0) AND NOT mergeNotPossible THEN
								nMoveState[nForCounter] := 70;
							END_IF 
				//	END_IF
				70:  //merge with gap zero
					//issue commmand to sync 
					IF  directMerge THEN 
						fbMover[nForCounter].P_Dynamics.SetValuesVADJ(stMoverConfigNormal.velo,stMoverConfigNormal.Accel,stMoverConfigNormal.Decel,stMoverConfigNormal.Jerk);
						fbMover[nForCounter].MoveOnTrack(track:= GVL_Mc.MC_Tracks[E_TrackNum.Main], targetPos:= GVL_Mc.MC_Tracks[E_TrackNum.Main].GetLength()-500, gap:= stMoverConfigNormal.MoverGap, velo:= stMoverConfigNormal.velo);

						nMoveState[nForCounter] := 10; 
					ELSIF moverInFront <>0 THEN 
						fbMover[nForCounter].P_Dynamics.SetValuesVADJ(stMoverConfigNormal.velo,stMoverConfigNormal.Accel,stMoverConfigNormal.Decel,stMoverConfigNormal.Jerk);
						masterSyncPos := GVL_Mc.MC_Tracks[E_TrackNum.Big].GetLength()-2500;
						masterPosAtSync := Mover[moverInFront].MoverPos; 
						followSyncPos := GVL_Mc.MC_Tracks[E_TrackNum.Small].GetLength()-stMoverConfigNormal.MoverGap-2500;
						followerPosAtSync :=Mover[nForCounter].MoverPos; 
						fbMover[nForCounter].SyncToOtherMover( 
							masterSyncPos := masterSyncPos,
							masterTrack := GVL_Mc.MC_Tracks[E_TrackNum.Big],
							followerSyncPos := followSyncPos,
							followerTrack := GVL_Mc.MC_Tracks[e_TrackNum.Small],
							PlanarMoverToFollow := fbMover[moverInFront].P_PlanarMover,
							velo:= stMoverConfigNormal.velo);
							nMoveState[nForCounter] := 80; 
						// reduce the gap of the leading mover 
						fbMover[moverInFront].MoveOnTrack(track:= GVL_Mc.MC_Tracks[E_TrackNum.Main], targetPos:= GVL_Mc.MC_Tracks[E_TrackNum.Main].GetLength()-500, gap:= 0, velo:= stMoverConfigNormal.velo);

					END_IF 
					
				80: // wait for in Sync 
					IF fbMover[nForCounter].P_SyncFeedback.Active AND MOver[moverInFront].TrackID =  GVL_Mc.MC_Tracks[E_TrackNum.Big].MCTOPLC_STD.TrackOID THEN // actively syncing calculate distance from mover 
						followerToEndOfTrack := fbMover[nForCounter].distToEndOfTrack; 
						leaderToEndofTrack := fbMover[moverInFront].distToEndOfTrack; 
						distToMoverInFront := followerToEndOfTrack - leaderToEndofTrack; 
					ELSE 
						followerToEndOfTrack := 0; 
						leaderToEndofTrack := 0; 
						distToMoverInFront := 0;
					END_IF
					IF fbMover[nForCounter].P_SyncFeedback.inSync OR  MOver[nForCounter].TrackID =  GVL_Mc.MC_Tracks[E_TrackNum.Main].MCTOPLC_STD.TrackOID THEN 
						nMoveState[nForCounter] := 10;
						IsMoverCommandedInShortcut :=FALSE;
					ELSIF	fbMover[nForCounter].P_SyncFeedback.Error THEN
						nMoveState[nForCounter] := 60;
					END_IF 
					
				END_CASE
		
		END_FOR

		rt_InitStop(CLK := HMI_StopCmd OR NOT GVL_Mc.HWStop);
		IF rt_InitStop.Q AND NOT bStopSequence THEN
			bStopSequence := TRUE;
		END_IF
		IF bStopSequence AND NOT(IsMoverInBlockingArea) THEN
			nCase := 110;
			bStopSequence := FALSE;
		END_IF
		
		110:
			N:= nNumMovers;
			FOR nForCounter:=1 TO nNumMovers DO		
				aStopPositions[nForCounter] := fbMover[nForCounter].XtsXlMover.GetSimulatedStartUpPosition(0);
				N := N -1;
			END_FOR
			nCase := 120;
		
		120:	
			nActStopPos := UDINT_TO_UINT(nMoverCount-nNumMovers+1);
			FOR nForCounter:=1 TO nNumMovers DO
				fbMover[nForCounter].P_Dynamics.SetValuesVADJ(stMoverConfigNormal.velo,stMoverConfigNormal.Accel,stMoverConfigNormal.Decel,stMoverConfigNormal.Jerk);
				nMoveState[nForCounter] := 0;
				fbMover[nForCounter].MoveOnTrack(track:= GVL_Mc.MC_Tracks[E_TrackNum.Main], targetPos:= 300, gap:= stMoverConfigNormal.MoverGap, velo:= 1000);
			END_FOR

			nCase:= 130; 
		130:
			FOR nForCounter:=1 TO nMoverCount - (nMoverCount -nNumMovers)  DO
				CASE nMoveState[nForCounter] OF
					0:								
						IF Mover[nForCounter].MoverPos < 300 AND  Mover[nForCounter].TrackID = GVL_Mc.MC_Tracks[E_TrackNum.main].MCTOPLC_STD.TrackOID THEN
							fbMover[nForCounter].MoveOnTrack(track:= GVL_Mc.MC_Tracks[E_TrackNum.Main], targetPos:= aStopPositions[nActStopPos], gap:= stMoverConfigNormal.MoverGap, velo:= 1000);

							nActStopPos := nActStopPos + 1;
							nMoveState[nForCounter] := 10;
						END_IF
				END_CASE
			END_FOR
		
			bAllDone := TRUE;
			FOR nForCounter:=1 TO nNumMovers DO
				IF NOT(MoverFeedback[nForCounter].Done OR MoverFeedback[nForCounter].Error) THEN
					bAllDone := FALSE;
					EXIT;
				END_IF
			END_FOR
			
			IF bAllDone THEN
				nCase := 150;
			END_IF
		
		140:
			FOR nForCounter:=1 TO nNumMovers DO
				fbMover[nForCounter].P_PlanarMover.Halt(MoverFeedback[nForCounter], haltDynamics);
			END_FOR	
			
			nCase := 145;
			
		145:
			bAllDone := TRUE;
			FOR nForCounter:=1 TO nNumMovers DO
				IF NOT(MoverFeedback[nForCounter].Done OR MoverFeedback[nForCounter].Error) THEN
					bAllDone := FALSE;
					EXIT;
				END_IF
			END_FOR
			
			IF bAllDone THEN
				nCase := 150;
			END_IF
		
		//Disable
		150:
			MoverStopDone := TRUE;
			FOR nForCounter:=1 TO nNumMovers DO
				fbMover[nForCounter].P_PlanarMover.Disable(MoverFeedback[nForCounter]);
			END_FOR
				
			nCase := 0;
END_CASE

bMagnetOn := FALSE;
FOR nForCounter:=1 TO nNumMovers DO
	
	IF  fbMover[nForCounter].XtsXlMover.GetPositionInfo_trackObjectId(0) = XtsShortcutOid AND (IsBetween(fbMover[nForCounter].XtsXlMover.GetPositionInfo_trackPosition(0), SwitchConfig.MagnetStartPosition - (stMoverConfigNormal.Velo*0.045), SwitchConfig.MagnetEndPosition)) THEN
		bMagnetOn := TRUE;
	END_IF
END_FOR

IF SwitchConfig.UseNominalCurrentVeloSetpoints THEN
	SwitchStatus.CurrentTheorOutputMax := SwitchConfig.SwitchCurrentNominal;	
ELSE
	SwitchStatus.CurrentTheorOutputMax := ((SwitchConfig.MagnetConfig.CurrentFunctionCoeffA*(((stMoverConfigNormal.Velo/1000)*(stMoverConfigNormal.Velo/1000))))+(SwitchConfig.MagnetConfig.CurrentFunctionCoeffB*(stMoverConfigNormal.Velo/1000))+SwitchConfig.MagnetConfig.CurrentFunctionCoeffC);	
END_IF

SwitchStatus.CurrentActualOutput := F_MapLReal(
	x:= MagnetFdbkValue, 
	in_min:= 0, 
	in_max:= 32767, 
	out_min:= 0, 
	out_max:= 54);

IF bMagnetOn AND NOT Fault THEN
	MagnetValue := TO_INT(SwitchStatus.CurrentTheorOutputMax*1310);
ELSE
 	MagnetValue := 0;
END_IF

FP_Counter(clk:=bMagnetOn);

IF FP_Counter.Q THEN
	Switchcounter := Switchcounter+1;

END_IF

//distanceMonitoring of Mover 1 when on the big track 
IF Mover[1].TrackID = GVL_Mc.MC_Tracks[E_TrackNum.Main].MCTOPLC_STD.TrackOID THEN //calculate out how far it is to the mover in front 
	IF MOver[stMergeConfig.moverInFront].MoverPos -  Mover[1].MoverPos > 10 THEN 
		stMergeConfig.mover1FollowDist := MOver[stMergeConfig.moverInFront].MoverPos -  Mover[1].MoverPos;
	END_IF   
END_IF

END_PROGRAM

// ---- POUs/FB_TrackObject.TcPOU
FUNCTION_BLOCK FB_TrackObject
// for a track/part this block keeps a list of the movers in order with their positions on a track

VAR_INPUT
	TrackID: OTCID;
	iMover	:REFERENCE TO ARRAY[1..nMoverCount] OF I_Mover;
	trackLength : LREAL;// this should be a loookup but I don't know how to look it up so I'm going to pass it externally 
END_VAR

VAR_OUTPUT
	bBusy: BOOL;
	bDone: BOOL;
	bError: BOOL;
	bInit: BOOL;
	ipResultMessage: I_TcMessage := fbResult;
	moverIDs : ARRAY[1..nMoverCount] OF UDINT;
END_VAR

VAR
	nNumMoversThisTrack: UDINT; //numberofMovers currently on this track
	nMoverList: ARRAY [1..nMoverCount] OF OTCID; //list of movers currently on the track 

	distToNextMover : ARRAY[1..nMoverCount] OF LREAL;  
END_VAR

VAR

	fbResult: FB_TcMessage;
	_ipComObject: ITComObject;
	PID_MOverList				: PTCID := 16#05030149;
	PID_NumMover				: PTCID := 16#050300C5;
END_VAR

IF NOT bInit THEN
	IF GetComObject(nObjectId:=TrackID) THEN
		bInit:=TRUE;
	END_IF
	RETURN;
END_IF

METHOD CyclicUpdate : BOOL
VAR_INPUT
END_VAR

VAR
	J: UDINT;
	I: UDINT;
END_VAR
IF bInit THEN 
	GetNumMovers(); 
	GetMoverList(); 
END_IF 
MEMSET(ADR(moverIDs),0,SIZEOF(moverIDs)); // have to clear the list 
FOR J := 1 TO nNumMoversThisTrack DO  
	FOR I := 1 TO nNumMovers DO  
		IF iMover[I].MoverOTCID = nMoverList[J] THEN 
			moverIDs[J] := I; 
		END_IF
	END_FOR
END_FOR
FOR I := 1 TO nNumMoversThisTrack DO 
	IF I <= nNumMoversThisTrack -1 THEN
		distToNextMover[I] := fbMover[moverIDs[I+1]].distToEndOfTrack - fbMover[moverIDs[I]].distToEndOfTrack;
	ELSIF I = nNumMoversThisTrack THEN
		distToNextMover[I] := trackLength - fbMover[moverIDs[I]].distToEndOfTrack;
	END_IF
END_FOR
END_METHOD

METHOD findMergePosition : BOOL
VAR_INPUT
	mergeSyncCommandPos : LREAL;
	spaceToMerge :LREAL; 
END_VAR
VAR_OUTPUT 
	nMoverToFollow: UDINT; 
	mergeWithoutFollow : BOOL; 
	mergeNotPossible : BOOL; 
END_VAR
VAR_INST 
	I: UDINT;
	moverInMerge: UDINT;
END_VAR
mergeNotPossible := TRUE; 
mergeWithoutFollow:=FALSE;
nMoverToFollow := 0; 
moverInMerge := 0;
// do not get fancy,  go through the list find all the distances between
//cyclic update finds builds a list of moers on the track and their spaceing 

IF nNumMoversThisTrack = 0  THEN // if there's no movers on the track we can just merge 
	mergeWithoutFollow := TRUE;
	mergeNotPossible := FALSE; 
ELSE
	// find a mover to follow starting at sync position look for a space to merge sized hole 
	FOR I := 1 TO nNumMoversThisTrack DO 
		IF fbMover[moverIDs[I]].distToEndOfTrack > mergeSyncCommandPos THEN // this mover is a potentialmover to follow 
			IF distToNextMover[I] > spaceToMerge THEN // follow this mover 
				nMoverToFollow := moverIDs[I]; //yes follow this mover 
				mergeNotPossible := FALSE; // the merge is possible 
				EXIT ; //get out of the loop we want the first one 
			END_IF
		END_IF
	END_FOR 
END_IF
IF mergeNotPossible THEN 
	nMoverToFollow := 0; 
END_IF
END_METHOD

METHOD GetComObject : BOOL
VAR_INPUT
	nObjectId: OTCID;
END_VAR
IF FW_ObjMgr_GetObjectInstance(	oid		:= nObjectId, 
								iid		:= TC_GLOBAL_IID_LIST.IID_ITComObject, 
								pipUnk	:= ADR(_ipComObject)) = 0
THEN
	GetComObject := TRUE;
END_IF
END_METHOD

METHOD GetMoverList : BOOL
VAR
	nData 			: UDINT := SIZEOF(nMoverList);
	pData 			: PVOID := ADR(nMoverList);
	stEventEntry	: TcEventEntry;
	pstEventEntry	: REFERENCE TO TcEventEntry REF= stEventEntry;
END_VAR
VAR_INST
	hResult : HRESULT;
END_VAR
bError := FALSE;

IF _ipComObject <> 0 THEN 
	 hResult := 	_ipComObject.TcgetObjPara(		pid := PID_MOverList,
													nData := nData,
													pData := pData,
													pgp := 0); 	
	IF hResult = 0 THEN
		GetMoverList := TRUE;
	ELSE
		HRESULTAdsErr_TO_TcEventEntry(hResult,stEventEntry);
		IF NOT fbResult.EqualsToEventEntryEx( stOther := stEventEntry) THEN
			fbResult.CreateEx(stEventEntry, 0);
			fbResult.Send(0);
			fbResult.Release();
		END_IF
		bError := TRUE;
	END_IF							
END_IF
END_METHOD

METHOD GetNumMovers : BOOL
VAR
	stEventEntry: TcEventEntry;
	pstEventEntry: REFERENCE TO TcEventEntry := stEventEntry;
	nData 			: UDINT := SIZEOF(nNumMoversThisTrack);
	pData 			: PVOID := ADR(nNumMoversThisTrack);
END_VAR

VAR_INST
	hResult : HRESULT;
END_VAR
bError := FALSE;

IF _ipComObject <> 0 THEN 	
	nData := SIZEOF(nNumMoversThisTrack);
	pData  := ADR(nNumMoversThisTrack);

	 hResult := 	_ipComObject.TcGetObjPara(		pid := PID_NumMover,
													nData := nData,
													pData := pData,
													pgp := 0); 	
													
	IF hResult = 0 THEN
		GetNumMovers := TRUE;
	ELSE
		HRESULTAdsErr_TO_TcEventEntry(hResult,stEventEntry);
		IF NOT fbResult.EqualsToEventEntryEx( stOther := stEventEntry) THEN
			fbResult.CreateEx(stEventEntry, 0);
			fbResult.Send(0);
			fbResult.Release();
		END_IF
		bError := TRUE;
	END_IF							
END_IF
END_METHOD

END_FUNCTION_BLOCK

// ---- POUs/IsBetween.TcPOU
FUNCTION IsBetween : BOOL
VAR_INPUT
	value: 	LREAL;
	minV:	LREAL;
	maxV:	LREAL;
END_VAR
VAR
END_VAR

IsBetween := value > minV AND value < maxV;

END_FUNCTION

// ---- XlMover/POUs/FB_Mover.TcPOU
{attribute 'no_assign'}
FUNCTION_BLOCK FB_Mover IMPLEMENTS I_Mover
VAR_INPUT
END_VAR
VAR_OUTPUT
END_VAR
VAR
	fbPlanarMover : MC_PlanarMover;
	fbPlanarFeedback: MC_PlanarFeedback;
	CmdFeedback :  XtsCommandFeedback;
	extrabyte : BYTE; 
	_bIsInitialized: BOOL;
	ipXtsMover:   I_XtsXlMover1;
	ipXtsProcessingUnit:  I_XtsProcessingUnit1;
	trackTrail: MC_PlanarTrackTrail;
	nextMcTrackOid: OTCID;
	stMoveOnTrackOptions: ST_MoveOnTrackOptions;
	_stDynamics: DynamicConstraint_PathXY;
	_TargetTrack : UDINT;
	_ReWork : BOOL;
	partConfig1: UINT;
	SyncMoverFeedback: Tc3_Mc3PlanarMotion.MC_PlanarFeedbackGearInPosOnTrackWithMasterMover;
	_InSync :BOOL; 
	options: Tc3_Mc3PlanarMotion.ST_GearInPosOnTrackWithMasterMoverOptions;
	syncTrail : MC_PlanarTrackTrail;
	_PositionOnTrack : LREAL;
	_Track : OTCID; 
	_distToEndOfTrack : LREAL;

END_VAR

METHOD CycleUpdate : BOOL
VAR_INPUT
END_VAR
VAR 
	_trackEnum: e_TrackNum;
END_VAR
IF NOT _bIsInitialized THEN
	RETURN;
END_IF

fbPlanarMover.GetTrackTrailInformation(trackTrail);
_PositionOnTrack := fbPlanarMover.MCTOPLC.SETONTRACK.SetPos;
IF fbPlanarMover.MCTOPLC.SETONTRACK.TrackOID<>0 THEN 
	_Track := fbPlanarMover.MCTOPLC.SETONTRACK.TrackOID;
	_trackEnum := F_GetTrackEnum(fbPlanarMover.MCTOPLC.SETONTRACK.TrackOID); 
	_distToEndOfTrack := GVL_Mc.MC_Tracks[_trackEnum].GetLength()-_PositionOnTrack;
END_IF

fbPlanarMover.Update();


fbPlanarFeedback.Update();
SyncMoverFeedback.Update(); 


UpdateXtsTrack();
END_METHOD

PROPERTY distToEndOfTrack : Lreal
GET
distToEndOfTrack := _distToEndOfTrack;
END_GET
END_PROPERTY

METHOD Init : BOOL
VAR_INPUT

	XtsMover:   I_XtsXlMover1;
	XtsProcessingUnit :  I_XtsProcessingUnit1;
END_VAR



ipXtsMover:= XtsMover;
ipXtsProcessingUnit :=  XtsProcessingUnit;

stMoveOnTrackOptions.direction := MC_Direction.mcDirectionPositive;
stMoveOnTrackOptions.gapMode := MC_GAP_MODE_ON_TRACK.Fast1D;
stMoveOnTrackOptions.gap:= 800;

syncTrail.AddTrack(track:= GVL_Mc.MC_Tracks[E_TrackNum.Small]); 
syncTrail.AddTrack(track:= GVL_Mc.MC_Tracks[E_TrackNum.Main]); 


//_stDynamics.SetValuesVADJ(500, 4000, 4000, 10000);

_bIsInitialized := TRUE;
Init := TRUE;
END_METHOD

METHOD JoinNearestTrack : BOOL


VAR_INST
	nForCounter: UINT;
	mcTrackOid: OTCID;
	partOid: OTCID;
	cmdFeedback					: 	XtsCommandFeedback;
	objectInfo: PlanarObjectInfo;
END_VAR
partOid := ipXtsMover.GetPositionInfo_partObjectId(cmdFeedback);

IF partOid = 0 THEN
	RETURN;
END_IF

IF cmdFeedback.IsDone THEN
	mcTrackOid := ipXtsProcessingUnit.XlPartWithOid(partOid, cmdFeedback).GetMcTrackOid(cmdFeedback);
	
	FOR nForCounter := 1 TO GVL_MC.nTrackCount DO
		objectInfo := GVL_MC.Mc_Tracks[nForCounter].GetPlanarObjectInfo();
		IF objectInfo.Id = mcTrackOid THEN
			fbPlanarMover.JoinTrack(fbPlanarFeedback, GVL_MC.Mc_Tracks[nForCounter], _stDynamics, 0); 
			RETURN;
		END_IF
	END_FOR
END_IF
END_METHOD

METHOD LeaveSystemAt : BOOL
VAR_INPUT
	ConnectionOut: REFERENCE TO MC_PlanarTrackConnectionOut;
END_VAR
fbPlanarMover.LeaveSystemAt(fbPlanarFeedback, ConnectionOut,  _stDynamics,0);
END_METHOD

METHOD MoveOnTrack : BOOL
VAR_INPUT
	
	track: REFERENCE TO MC_PlanarTrack;	
	targetPos: LREAL;
	gap : LREAL; 
	velo : LREAL; 
END_VAR
stMoveonTrackOptions.gap := gap; 

fbPlanarMover.MoveOnTrack(
	commandFeedback:= fbPlanarFeedback, 
	targetTrack:= track, 
	targetPositionOnTrack:= targetPos, 
	constraint:= _stDynamics, 
	options:= stMoveOnTrackOptions);
END_METHOD

PROPERTY MoverOTCID : OTCID
GET
MoverOTCID := fbPlanarMover.MCTOPLC.STD.MoverOID;
END_GET
SET
END_SET
END_PROPERTY

PROPERTY MoverStopped : BOOL
GET
MoverStopped := (fbPlanarMover.MCTOPLC.SETONTRACK.SetVelo < 20);
END_GET
SET
END_SET
END_PROPERTY

PROPERTY P_Dynamics : REFERENCE TO DynamicConstraint_PathXY;
GET

P_Dynamics REF= _stDynamics;
END_GET
SET // PUBLIC
_stDynamics := P_Dynamics;
END_SET
END_PROPERTY

PROPERTY P_IsInitialized : bool
GET
P_IsInitialized := _bIsInitialized;
END_GET
END_PROPERTY

PROPERTY P_PlanarFeedback : REFERENCE TO MC_PlanarFeedback
GET
P_PlanarFeedback REF= fbPlanarFeedback;
END_GET
END_PROPERTY

PROPERTY P_PlanarMover :   REFERENCE TO  MC_PlanarMover
GET
P_PlanarMover REF= fbPlanarMover;
END_GET
END_PROPERTY

PROPERTY P_SyncFeedback :  REFERENCE TO MC_PlanarFeedbackGearInPosOnTrackWithMasterMover
GET
P_SyncFeedback REF= SyncMoverFeedback;
END_GET
END_PROPERTY

PROPERTY P_TargetTrack : UDINT
GET
P_TargetTrack := _TargetTrack ;
END_GET
SET
_TargetTrack := P_TargetTrack;
END_SET
END_PROPERTY

PROPERTY Rework : BOOL
GET
Rework := _Rework;
END_GET
SET
_Rework := Rework;
END_SET
END_PROPERTY

METHOD SyncToOtherMover : BOOL
VAR_INPUT
	masterSyncPos : LREAL; // Position on the master track
	followerSyncPos : LREAL; // position on the follower track
	PlanarMoverToFollow: REFERENCE TO Tc3_Mc3PlanarMotion.MC_PlanarMover;
	masterTrack : REFERENCE TO Tc3_Mc3PlanarMotion.MC_PlanarTrack; 
	followerTrack : REFERENCE TO Tc3_Mc3PlanarMotion.MC_PlanarTrack; 
	velo : REFERENCE TO LREAL; 
END_VAR

VAR
	trail: Tc3_Mc3PlanarMotion.MC_PlanarTrackTrail;

END_VAR
Options.allowedSlaveSyncDirections := MC_SYNC_DIRECTIONS.Positive; 
options.directionMasterSyncPosition := MC_DIRECTION.mcDirectionNonModulo; 
options.directionSlaveSyncPosition := MC_DIRECTION.mcDirectionNonModulo;  
options.followMover := FALSE; 
options.gap := 0; // elimnate gap funciton 
options.inSyncToleranceDistance :=0; 
options.moduloToleranceMasterSyncPosition := 0; 
options.moduloToleranceSlaveSyncPosition := 0;  
_stDynamics.V := velo; 

fbPlanarMover.GearInPosOnTrackWithMasterMover(
	commandFeedback:=  SyncMoverFeedback , 
	masterMover:= PlanarMoverToFollow , 
	trackTrail:= syncTrail, // may need to give a trail maybe not
	masterSyncPosition:= masterSyncPos, 
	masterSyncPositionTrack:= MasterTrack , 
	slaveSyncPosition:= followerSyncPos, 
	slaveSyncPositionTrack:= followerTrack, 
	constraint:=_stDynamics , 
	options:=options );
END_METHOD

METHOD PUBLIC UpdateXtsTrack
VAR_INPUT
END_VAR
VAR_STAT
	nTrackCount: UINT;
	oid1: OTCID;
	oid2: OTCID;
	
	nForCounter: UINT;
	nPartConfigCount: UINT;
	
	partConfig1: OTCID;
	partConfig2: OTCID;
	
	mcTrackOid1: OTCID;
	mcTrackOid2: OTCID;
	trackOid: OTCID;
	
	nTrackTrailCount: UDINT;
	actTrackOid: OTCID;
	nIndexInTrail: UDINT;
END_VAR
nTrackTrailCount := trackTrail.TrackCount;
actTrackOid := fbPlanarMover.MCTOPLC.SETONTRACK.TrackOID;

IF nTrackTrailCount <= 1 THEN
	RETURN;
END_IF

FOR nForCounter := 1 TO UDINT_TO_UINT(nTrackTrailCount) DO
	oid1 := trackTrail.GetTrackOidAt(nForCounter);
	IF oid1 = actTrackOid THEN
		IF nForCounter < nTrackTrailCount THEN
			oid2 := trackTrail.GetTrackOidAt(nForCounter + 1);
			EXIT;
		ELSE
			RETURN; //last one ine track trail
		END_IF
	END_IF
END_FOR

IF oid2 = nextMcTrackOid AND   ipXtsMover.GetPositionInfo_partPosition(CmdFeedback) < 600THEN //no change
	RETURN;
END_IF

nTrackCount := ipXtsProcessingUnit.TrackCount();

FOR nForCounter := 1 TO nTrackCount DO
	nPartConfigCount := ipXtsProcessingUnit.Track(nForCounter, CmdFeedback).PartConfigCount(); 
	
	IF nPartConfigCount >= 2  THEN
		partConfig1 := ipXtsProcessingUnit.Track(nForCounter, CmdFeedback).GetPartConfigOidAt(1, 0);
		partConfig2 := ipXtsProcessingUnit.Track(nForCounter, CmdFeedback).GetPartConfigOidAt(2, 0);
//
		
		IF partConfig1 = 0 OR partConfig2 = 0 THEN
			CONTINUE;
		END_IF
		
		mcTrackOid1 := ipXtsProcessingUnit.XlPartWithOid(partConfig1, CmdFeedback).GetMcTrackOid(0);
		mcTrackOid2 := ipXtsProcessingUnit.XlPartWithOid(partConfig2, CmdFeedback).GetMcTrackOid(0);
		IF mcTrackOid1 = oid1 AND mcTrackOid2 = oid2   THEN
			trackOid := ipXtsProcessingUnit.Track(nForCounter, CmdFeedback).GetObjectId();
			ipXtsMover.SetActiveTrackObjectId(trackOid, CmdFeedback);
			
			IF CmdFeedback.IsDone THEN
				nextMcTrackOid := oid2;
			END_IF
			
			RETURN;
		END_IF
	END_IF
END_FOR
END_METHOD

PROPERTY XlProcessingUnit : I_XtsProcessingUnit1
GET
XlProcessingUnit := ipXtsProcessingUnit;
END_GET
END_PROPERTY

PROPERTY XtsComFeed : REFERENCE TO  XtsCommandFeedback
GET
XtsComFeed REF= CmdFeedback;
END_GET
END_PROPERTY

PROPERTY XtsXlMover : I_XtsXlMover1
GET
XtsXlMover := ipXtsMover;
END_GET
END_PROPERTY

END_FUNCTION_BLOCK

// ---- POUs/F_GetTrackEnum.TcPOU
FUNCTION F_GetTrackEnum : e_TrackNum
VAR_INPUT
	track : OTCID; 
END_VAR
VAR
END_VAR

IF GVL_Mc.MC_Tracks[E_TrackNum.Big].MCTOPLC_STD.TrackOID = track THEN 
	F_GetTrackEnum := E_TrackNum.Big; 
ELSIF 
	GVL_Mc.MC_Tracks[E_TrackNum.Small].MCTOPLC_STD.TrackOID = track THEN 
	F_GetTrackEnum := E_TrackNum.Small; 
ELSIF 
	GVL_Mc.MC_Tracks[E_TrackNum.Main].MCTOPLC_STD.TrackOID = track THEN 
	F_GetTrackEnum := E_TrackNum.Main; 
END_IF

END_FUNCTION

// ---- POUs/FB_PWM.TcPOU
FUNCTION_BLOCK FB_PWM
VAR_INPUT
	Torque: INT;
END_VAR

VAR
  	ModuleState AT %I* : UINT;
	
 	Control AT %Q* :  UINT;
 	TargetTorque AT %Q*: INT; 	

 	State  : INT := 1;
 	PwmTimer : ton;
END_VAR



CASE State OF 

	1: 
		Control := 6;
		IF ModuleState = 40 OR ModuleState = 33 THEN
			State := 5;
		END_IF
	5:
		Control := 128;
		IF ModuleState = 96 OR ModuleState = 33 OR ModuleState = 168 THEN
			State := 10;
		END_IF
	10:
		Control := 6;
		IF ModuleState = 33 THEN
			state := 15;
		END_IF	
	15:
		Control := 7;
		IF ModuleState = 35 OR ModuleState = 163 or ModuleState = 2083 THEN
			State := 20;
		END_IF	
	20:	
		Control := 15;
		IF ModuleState = 4135 OR ModuleState = 4263THEN
			state := 25;
		END_IF
	24:
	  //IF Torque = 0  THEN
			State := 25;
	//	END_IF	
		PwmTimer(in := FALSE,PT := T#30S);
	25:
		IF ModuleState = 40 THEN
			State := 5;
		END_IF
		
		IF Torque > 0 THEN
			TargetTorque := Torque ;
		ELSIF Torque = 0 AND TargetTorque > 0  THEN	
			TargetTorque :=  TargetTorque - REAL_TO_INT((INT_TO_REAL(TargetTorque)*0.07));
		END_IF	
		
		PwmTimer(in := TargetTorque > 300,PT := T#30S);
		IF PwmTimer.Q  THEN
			PwmTimer(in := FALSE,PT := T#30S);
			State := 35;
		END_IF 
	35:
		IF TargetTorque >0 THEN
			TargetTorque := TargetTorque -4;
		ELSIF 	TargetTorque = 0  THEN
				State := 24;
		END_IF	

END_CASE

END_FUNCTION_BLOCK

// ---- POUs/F_CalculateAccelTimeAndDistance.TcPOU
FUNCTION_BLOCK F_CalculateAccelTimeAndDistance
VAR_INPUT
	targetVelocity : LREAL; 
	Accel : LREAL; 
	Decel : LREAL; 
	Jerk : LREAL; 
	initialVelocity : LREAL; 
END_VAR
VAR_OUTPUT
	timeToReachVelocity : LREAL; 
	distanceTravelled : LREAL; 
END_VAR
VAR
	deltav: LREAL;
	timeAtAccel: LREAL;
	timeAtJerk: LREAL;
	velocityAfterJerk: LREAL;
	velocityChangeDuetoJerk: LREAL;
END_VAR

   // determine if the jerk allows for the acceleration to be reached or if the delta V is too small 
deltaV := targetVelocity - initialVelocity;

IF deltav * Jerk < Accel * Accel THEN 
	// accel lim is to high, jerk limited 
	timeAtAccel := 0; 
	timeAtJerk := SQRT(deltav/Jerk) ; 
ELSE // accel limit wil be reachead 
	timeAtJerk:= Accel/Jerk; 
	velocityChangeDuetoJerk := Accel * timeAtJerk/2.000; 
	velocityAfterJerk := initialVelocity +  velocityChangeDuetoJerk;
	timeAtAccel := (deltav - 2*velocityChangeDuetoJerk)/Accel; 
END_IF
 // calc time at max accel 
timeToReachVelocity := 2*timeAtJerk + timeAtAccel; 
distanceTravelled := initialVelocity * timeToReachVelocity + timeAtJerk *velocityChangeDuetoJerk *2 + timeAtAccel *velocityChangeDuetoJerk + Accel * timeAtAccel*timeAtJerk + 0.5* Accel* timeAtAccel*timeAtAccel;

END_FUNCTION_BLOCK

// ---- POUs/F_SearchTheBigTrackForAHole.TcPOU
FUNCTION_BLOCK F_SearchTheBigTrackForAHole
VAR_INPUT 
	resetSearch: BOOL;
	gapStartDistToEndOfSwitch : LREAL; 
	gapLength : LREAL; 	
END_VAR
VAR_IN_OUT 
	fbMover		:	ARRAY[1..GVL_mc.nMovercount] OF FB_Mover;
END_VAR
VAR_OUTPUT
	gapFound: BOOL;
	moverToFollow : UDINT; 
END_VAR
VAR
	I : UDINT; 
	nState: INT;
	trackPosGapStart  : LREAL; 
	trackPosGapEnd : LREAL;
	trackCollisionArea : LREAL; 
	moverTrackID: Global.GLOBAL.OTCID;
	lastMoverAfterGap: UDINT;
	closestAfterGap: LREAL;
	distanceAfterGap: LREAL;
	moverFound: BOOL;
END_VAR

IF resetSearch THEN 
//	nState := 0; 
END_IF

trackPosGapStart := GVL_Mc.MC_Tracks[E_TrackNum.Big].GetLength()-gapStartDistToEndOfSwitch; 
trackPosGapEnd := trackPosGapStart - gapLength; 
moverFound:= FALSE; 
gapFound := TRUE; 

//watch for a mover crossing the gap boundary and a free space behind it of 2m.  
FOR I:= 1 TO GVL_mc.nNumMovers DO 
	// Only evaluate Movers on the big track
	IF Mover[I].TrackID = GVL_Mc.MC_Tracks[E_TrackNum.Big].MCTOPLC_STD.TrackOID THEN  
		IF Mover[I].MoverPos > trackPosGapStart AND Mover[I].MoverPos < trackPosGapStart + 16  THEN 
			 moverFound := TRUE;  // there is a mover in the way, 
			 moverToFollow:=I; 
			 // since we are looking at each mover we want to look at each one only once 
		END_IF			
		//is a mover in the gap?   
		IF 	Mover[I].MoverPos < trackPosGapStart AND Mover[I].MoverPos > trackPosGapEnd THEN
			gapFound := FALSE; 						
		END_IF 
	END_IF 
END_FOR

gapFound :=  gapfound AND moverFound;


(*CASE nState OF
	0: //see if there is any mover in this range if there is no mover in this range go.  
		gapFound := TRUE; 
		lastMoverAfterGap := 0; 
		closestAfterGap := 10000; 
		FOR I:= 1 TO GVL_mc.nNumMovers DO 
			// Only evaluate Movers on the big track
			IF Mover[I].TrackID = GVL_Mc.MC_Tracks[E_TrackNum.Big].MCTOPLC_STD.TrackOID THEN  
				IF Mover[I].MoverPos < trackPosGapStart AND Mover[I].MoverPos > trackPosGapEnd  THEN 
					 gapFound := FALSE;  // there is a mover in the way, 
					 // since we are looking at each mover we want to look at each one only once 
				END_IF			
				//find last mover before gap 
				IF 	Mover[I].MoverPos > trackPosGapStart THEN
					distanceAfterGap :=  Mover[I].MoverPos - trackPosGapStart; 
					IF distanceAfterGap < closestAfterGap THEN 
						closestAfterGap := distanceAfterGap; 
						lastMoverAfterGap := I; 
					END_IF
				END_IF 
				IF closestAfterGap > 20 THEN // we want to follow a mover 
					gapFound:=FALSE; 
				END_IF
			END_IF 
		END_FOR
		moverToFollow := lastMoverAfterGap; 
END_CASE 		
*)

END_FUNCTION_BLOCK
